// TwinCAT 3 PLC project Untitled1
// ProgramVersion: 3.1.4024.0
// libraries:
//   Tc2_MC2, * (Beckhoff Automation GmbH)
//   Tc2_Standard, * (Beckhoff Automation GmbH)
//   Tc2_System, * (Beckhoff Automation GmbH)
//   Tc3_Module, * (Beckhoff Automation GmbH)
//   VisuDialogs, * (System)
//   VisuSymbols,3.5.10.0,System
// project tree:
//   / GlobalTextList.TcGTLO, PlcTask.TcTTO, Visualization Manager.TcVMO (not stored)
//   GVLs/ GVL.TcGVL
//   POUs/ AxisControl.TcPOU, MAIN.TcPOU
//   VISUs/ HMI.TcVIS
// real-time tasks:
//   TASK PlcTask: cycle T#10ms, priority 20, ADS port 350
// motion (NC):
//   TASK NC-Task 1 SAF: cycle T#2ms, priority 4, ADS port 501
//   TASK NC-Task 1 SVB: cycle T#10ms, priority 8, ADS port 511
//   AXIS Axis 1 (id 1)
//     Dynamic: Acceleration=120, Deceleration=120, Jerk=1000
//     Velo: SlowManual=20, FastManual=70, Maximum=150
//     OtherSettings: AllowMotionCmdToSlave=true
//     encoder EncType=1
//       EncPara: ScaleFactorNumerator=1
//         SoftEndMinControl: Enable=true, Range=-500
//         SoftEndMaxControl: Enable=true, Range=500
//     drive DrvType=5
//       Analog: VeloReferenz=100, TorqueSetpointScale=10, ScaleFactorActTorque=0.1
//       TimeComp: TaskDelayCycles=1
//     controller CtrType=1
//       CtrPara: PriorControlFactor=1
//         Observer: BandWidth=20
// variable links:
//   Untitled1/Untitled1 Instance <-> NC-Task 1 SAF/Axes/Axis 1
//     PlcTask Inputs/GVL.Axis.NcToPlc <-> Outputs/ToPlc
//     PlcTask Outputs/GVL.Axis.PlcToNc <-> Inputs/FromPlc

CONFIGURATION Untitled1
    RESOURCE PLC ON TwinCAT3
        TASK PlcTask(INTERVAL := T#10ms, PRIORITY := 20);
        PROGRAM MAIN WITH PlcTask : MAIN;
    END_RESOURCE
END_CONFIGURATION

// ---- GVLs/GVL.TcGVL
{attribute 'qualified_only'}
VAR_GLOBAL
	Axis : AXIS_REF;
END_VAR

// ---- POUs/MAIN.TcPOU
PROGRAM MAIN
VAR
	AxisControl : AxisControl;
	
END_VAR

AxisControl();
//AxisControl2();

END_PROGRAM

// ---- POUs/AxisControl.TcPOU
FUNCTION_BLOCK AxisControl
VAR_INPUT
END_VAR
VAR_OUTPUT
	//Position
	ActualPosition : LREAL;
	//Velocity
	ActualVelocity : LREAL;
END_VAR
VAR
	//Power
	McPower : MC_Power;
	McPowerEnable : BOOL;
	McPowerError : BOOL;
	AxisStatus : BOOL;
	//JOG
	McJog : MC_Jog;
	JogForward : BOOL;
	JogBackward : BOOL;

	//Relative
	McMoveRelative : MC_MoveRelative;
	ExecuteRelative : BOOL;
	RelativeDistance : LREAL;
	RelativeVelocity : LREAL;
	//Absolute
	McMoveAbsolute : MC_MoveAbsolute;
	ExecuteAbsolute : BOOL;
	AbsolutePosition : LREAL;
	AbsoluteVelocity : LREAL;
	//Velocity
	McMoveVelocity : MC_MoveVelocity;
	ExecuteVelocity : BOOL;
	Velocity : LREAL;
	//Home
	McHome: MC_Home;
	ExecuteHome : BOOL;
	HomeSensor : BOOL;
	//Stop
	McStop : MC_Stop;
	ExecuteStop : BOOL;
	//Halt
	McHalt: MC_Halt;
	ExecuteHalt : BOOL;
END_VAR

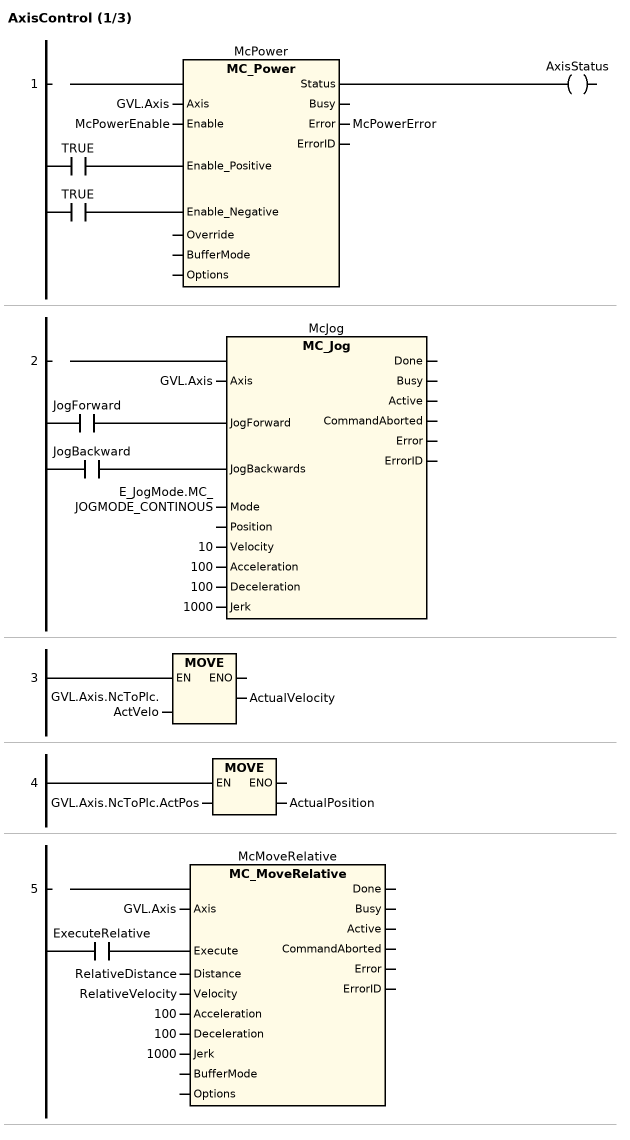
// NETWORK 1
McPower(
    Axis := GVL.Axis,
    Enable := McPowerEnable,
    Enable_Positive := TRUE,
    Enable_Negative := TRUE,
    Error => McPowerError); // MC_Power
AxisStatus := McPower.Status;

// NETWORK 2
McJog(
    Axis := GVL.Axis,
    JogForward := JogForward,
    JogBackwards := JogBackward,
    Mode := E_JogMode.MC_JOGMODE_CONTINOUS,
    Velocity := 10,
    Acceleration := 100,
    Deceleration := 100,
    Jerk := 1000); // MC_Jog

// NETWORK 3
ActualVelocity := GVL.Axis.NcToPlc.ActVelo;

// NETWORK 4
ActualPosition := GVL.Axis.NcToPlc.ActPos;

// NETWORK 5
McMoveRelative(
    Axis := GVL.Axis,
    Execute := ExecuteRelative,
    Distance := RelativeDistance,
    Velocity := RelativeVelocity,
    Acceleration := 100,
    Deceleration := 100,
    Jerk := 1000); // MC_MoveRelative

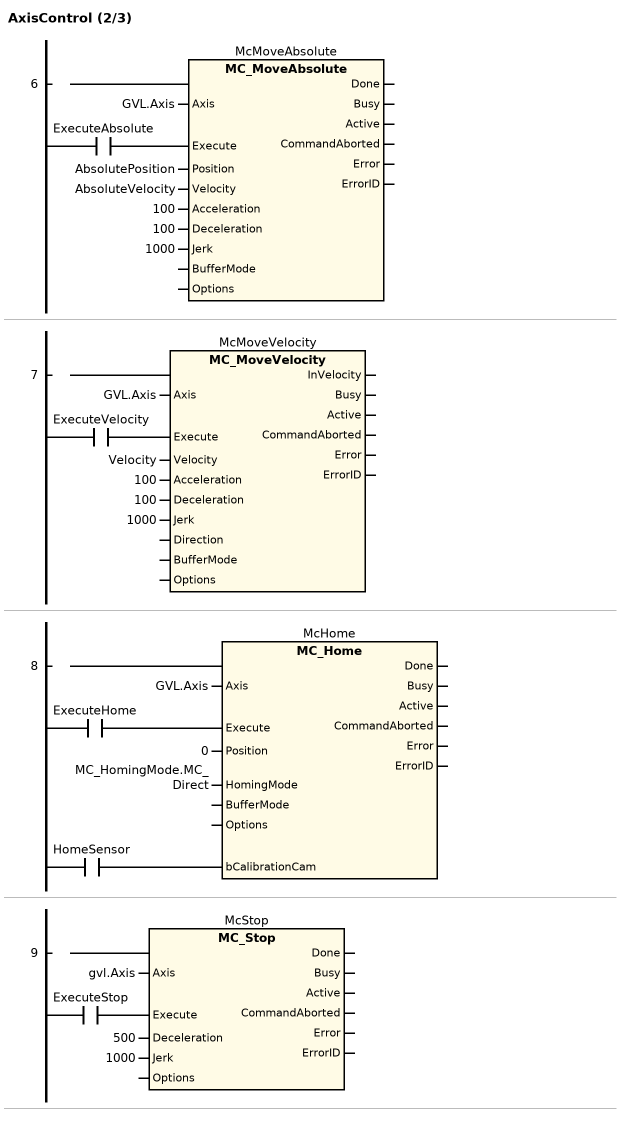
// NETWORK 6
McMoveAbsolute(
    Axis := GVL.Axis,
    Execute := ExecuteAbsolute,
    Position := AbsolutePosition,
    Velocity := AbsoluteVelocity,
    Acceleration := 100,
    Deceleration := 100,
    Jerk := 1000); // MC_MoveAbsolute

// NETWORK 7
McMoveVelocity(
    Axis := GVL.Axis,
    Execute := ExecuteVelocity,
    Velocity := Velocity,
    Acceleration := 100,
    Deceleration := 100,
    Jerk := 1000); // MC_MoveVelocity

// NETWORK 8
McHome(
    Axis := GVL.Axis,
    Execute := ExecuteHome,
    Position := 0,
    HomingMode := MC_HomingMode.MC_Direct,
    bCalibrationCam := HomeSensor); // MC_Home

// NETWORK 9
McStop(Axis := gvl.Axis, Execute := ExecuteStop, Deceleration := 500, Jerk := 1000); // MC_Stop

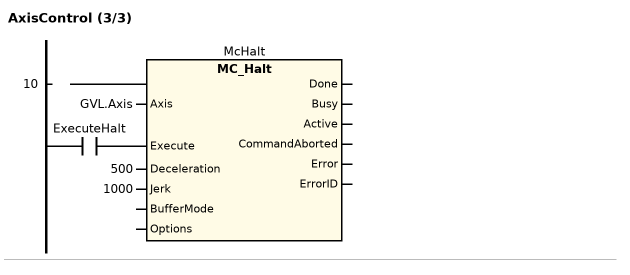
// NETWORK 10
McHalt(Axis := GVL.Axis, Execute := ExecuteHalt, Deceleration := 500, Jerk := 1000); // MC_Halt

END_FUNCTION_BLOCK

// ---- GlobalTextList.TcGTLO
TEXTLIST GlobalTextList
  489 = '%.0f'
  115 = 'Actual position'
  103 = 'Data'
  689 = 'Drive Control'
  693 = 'Drive enable'
  124 = 'Enter velocity'
  777 = 'Halt motion'
  326 = 'Jog+'
  694 = 'Jog-'
  95 = 'Manual control'
  679 = 'Manual motion'
  174 = 'Move absolute'
  964 = 'Move home'
  708 = 'Move relative'
  588 = 'Move velocity'
  468 = 'Power'
  536 = 'Stop motion'
  27 = 'Type absolute pos'
  85 = 'Type absolute velocity'
  97 = 'Type relative pos'
  81 = 'Type relative velocity'
  642 = 'Type velocity'
  655 = 'Velocity'
  341 = 'Vlamai'
END_TEXTLIST

// ---- VISUs/HMI.TcVIS
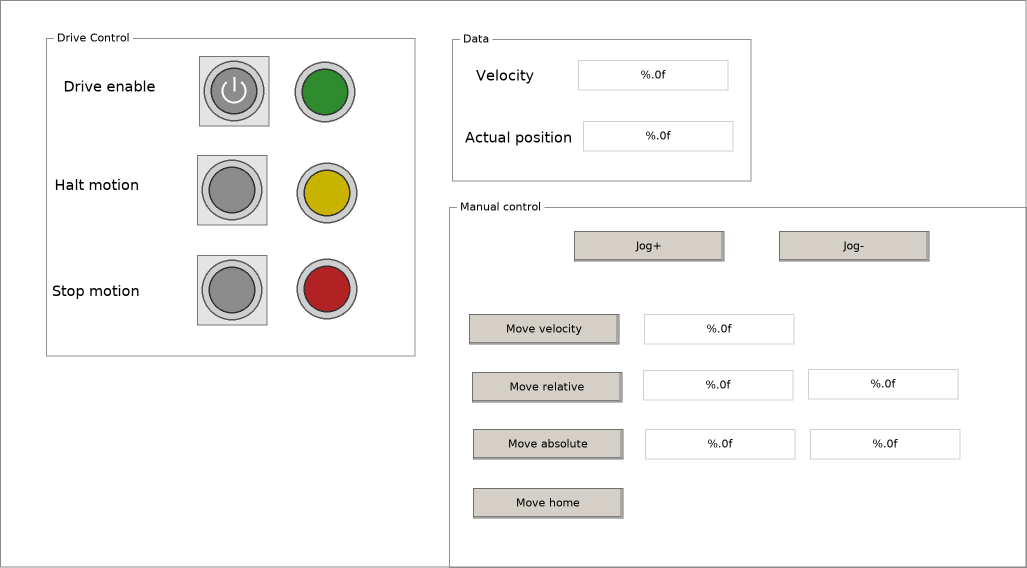
VISUALIZATION HMI  // 1027x568
    GroupBox (46,30 369x326), "Drive Control"
        PowerSwitch (153,26 70x70), variable: MAIN.AxisControl.McPowerEnable, behaviour: TOGGLE, style: Switch-PowerSwitch-Gray
        Lamp1 (244,27 70x70), variable: MAIN.AxisControl.AxisStatus, style: Lamp-Lamp1-Green
        PushSwitch (151,125 70x70), variable: MAIN.AxisControl.ExecuteHalt, behaviour: TOGGLE, style: Switch-PushSwitch-Gray
        PushSwitch (151,225 70x70), variable: MAIN.AxisControl.ExecuteStop, behaviour: TOGGLE, style: Switch-PushSwitch-Gray
        Lamp1 (246,128 70x70), variable: MAIN.AxisControl.McHalt.Done, style: Lamp-Lamp1-Yellow
        Lamp1 (246,224 70x70), variable: MAIN.AxisControl.McStop.Done, style: Lamp-Lamp1-Red
    Label (22,170 150x30), "Halt motion"
    Label (21,276 150x30), "Stop motion"
    Label (44,66 131x41), "Drive enable"
    GroupBox (452,31 299x150), "Data"
        Label (6,32 94x25), "Velocity"
        Textfield (126,29 150x30), "%.0f", text variable: MAIN.AxisControl.ActualVelocity
        Label (11,95 111x23), "Actual position"
        Textfield (131,90 150x30), "%.0f", text variable: MAIN.AxisControl.ActualPosition
    GroupBox (449,199 578x369), "Manual control"
        Button (125,32 150x30), "Jog+"
            OnMouseDown: toggle MAIN.AxisControl.JogForward
        Button (330,32 150x30), "Jog-"
            OnMouseDown: toggle MAIN.AxisControl.JogBackward
        Button (20,115 150x30), "Move velocity"
            OnMouseDown: toggle MAIN.AxisControl.ExecuteVelocity
        Textfield (195,115 150x30), "%.0f", tooltip "Type velocity", text variable: MAIN.AxisControl.Velocity
            OnMouseClick: write the text variable via Edit, min 0, max 50
        Button (23,173 150x30), "Move relative"
            OnMouseDown: toggle MAIN.AxisControl.ExecuteRelative
        Textfield (194,171 150x30), "%.0f", tooltip "Type relative pos", text variable: MAIN.AxisControl.RelativeDistance
            OnMouseClick: write the text variable via Edit
        Button (24,230 150x30), "Move absolute"
            OnMouseDown: toggle MAIN.AxisControl.ExecuteAbsolute
        Textfield (196,230 150x30), "%.0f", tooltip "Type absolute pos", text variable: MAIN.AxisControl.AbsolutePosition
            OnMouseClick: write the text variable via Edit
        Button (24,289 150x30), "Move home"
            OnMouseDown: toggle MAIN.AxisControl.ExecuteHome
        Textfield (359,170 150x30), "%.0f", tooltip "Type relative velocity", text variable: MAIN.AxisControl.RelativeVelocity
            OnMouseClick: write the text variable via Edit
        Textfield (361,230 150x30), "%.0f", tooltip "Type absolute velocity", text variable: MAIN.AxisControl.AbsoluteVelocity
            OnMouseClick: write the text variable via Edit
END_VISUALIZATION
